// TIA Portal V19 export
TYPE "LEXCHANGETRAY_typeConstraintRollerEm_deliver_interface"
// stored: Access Published
   STRUCT
      init : Bool;
      roller : "LEXCHANGETRAY_typeConstraintRollerEm_toRollerDeliver";
      constraintWorkstation { S7_SetPoint := 'True'} : "LEXCHANGETRAY_typeConstraintRollerEm_toConstraintWorkstationDeliver";
      handlingXyz { S7_SetPoint := 'True'} : "LEXCHANGETRAY_typeConstraintRollerEm_toHandlingXyzDeliver";
   END_STRUCT;
END_TYPE
